// TIA Portal V20 export
// export: Created 2026-07-10T11:12:27.281158Z, ExportSetting WithDefaults, DisplayName Totally Integrated Automation Portal, DisplayVersion V20, DisplayName TIA Portal Openness, DisplayVersion V20, DisplayName TIA Portal Version Control Interface, DisplayVersion V20, DisplayName STEP 7 Professional, DisplayVersion V20, DisplayName STEP 7 Safety, DisplayVersion V20, DisplayName WinCC Basic/Comfort/Advanced, DisplayVersion V20, DisplayName WinCC Unified, DisplayVersion V20
DATA_BLOCK "AIHandler_DB"   // DB4
VERSION : 0.1
// stored: AutoNumber true, DBAccessibleFromOPCUA true, InstanceOfName AIHandler, InstanceOfType FB
"AIHandler"
   // VAR_INPUT
   //    Value : Real := 0.0;
   //    ValueMin : Real := 0.0;
   //    ValueMax : Real := 0.0;
   //    ValueOffset : Real := 0.0;
   //    OutputMin : Real := 0.0;
   //    OutputMax : Real := 0.0;
   //    TimeBase : Time := T#1S;
   // END_VAR
   // VAR_OUTPUT
   //    Output : Real := 0.0;
   //    Error : Bool := FALSE;
   // END_VAR
   // VAR
   //    ConvertedValue : Real := 0.0;
   //    TON1 { S7_SetPoint := 'True'} : TON_TIME;
   //    DelayTON { S7_SetPoint := 'True'} : TON_TIME;
   //    FilterArray : Array[0..199] of Real;
   //    FilterTime : Time := T#0MS;
   //    i : Int := 0;
   //    sum : Real := 0.0;
   //    FilteredValue : Real := 0.0;
   //    one : Bool := FALSE;
   // END_VAR
BEGIN
   TON1.PT := T#0MS;
   TON1.IN := FALSE;
   DelayTON.PT := T#0MS;
   DelayTON.IN := FALSE;
   FilterArray[0..199] := 0.0;
END_DATA_BLOCK
